PROGRAM PRG_Static
VAR
	k: INT;
	l: INT;
	m: INT;
END_VAR

	stat_scalar_BOOL	:= TRUE;
	stat_scalar_I1		:= 1;	
	stat_scalar_UI1		:= 1;	
	stat_scalar_I2 		:= 1;		
	stat_scalar_UI2		:= 1;	
	stat_scalar_I4		:= 1;	
	stat_scalar_UI4		:= 1;	
	stat_scalar_I8		:= 1;	
	stat_scalar_UI8		:= 1;	
	stat_scalar_BYTE	:= 1;	
	stat_scalar_WORD	:= 1;	
	stat_scalar_DWORD	:= 1;	
	stat_scalar_LWORD	:= 1;				
	stat_scalar_R4		:= 1.0;				
	stat_scalar_R8		:= 1.0;				
	stat_scalar_BSTR	:= 'Hello World';
	stat_scalar_WSTRING	:= "Hello World";
	stat_scalar_DT		:= DT#1972-03-29-00:00:00;
	stat_scalar_DATE 	:= DATE#1972-03-29;
	stat_scalar_TOD		:= TOD#12:00:00;	
	stat_scalar_TIME	:= T#1S;	

	GVL_structures.StructuredType1.a 			:= 42;
	GVL_structures.StructuredType1.b			:= 42;
	GVL_structures.StructuredType1.x			:= E_Enum_1.THREE;
	GVL_structures.StructuredType1.str			:= 'Hello World';

	GVL_structures.StructuredType2.c1.a			:= 42;
	GVL_structures.StructuredType2.c1.b			:= 42;
	GVL_structures.StructuredType2.c1.x			:= E_Enum_1.THREE;
	GVL_structures.StructuredType2.c1.str		:= 'Hello World';
	GVL_structures.StructuredType2.s_5			:= 'Hello';
	GVL_structures.StructuredType2.s_3			:= 'Hel';
	FOR k:= 0 TO 5 DO
		GVL_structures.StructuredType2.cArr[k].a:= 42;
		GVL_structures.StructuredType2.cArr[k].b:= 42;
		GVL_structures.StructuredType2.cArr[k].x:= E_Enum_1.THREE;
		GVL_structures.StructuredType2.cArr[k].str:= 'Hello World'; 
	END_FOR	
	GVL_structures.StructuredType2.e			:= E_Enum_1.THREE;
	FOR k:= 0 TO 100 DO
		GVL_structures.StructuredType2.iArr[k] := 42;
	END_FOR
	
	GVL_structures.StructuredType8.stComplex.a			:= 42;
	GVL_structures.StructuredType8.stComplex.b			:= 42;
	GVL_structures.StructuredType8.stComplex.x			:= E_Enum_1.THREE;
	GVL_structures.StructuredType8.stComplex.str		:= 'Hello World';
	GVL_structures.StructuredType8.strString5			:= 'Hello';
	GVL_structures.StructuredType8.strString3			:= 'Hel';
	FOR k:= 0 TO 1 DO
		GVL_structures.StructuredType8.arrComplex[k].a:= 42;
		GVL_structures.StructuredType8.arrComplex[k].b:= 42;
		GVL_structures.StructuredType8.arrComplex[k].x:= E_Enum_1.THREE;
		GVL_structures.StructuredType8.arrComplex[k].str:= 'Hello World'; 
	END_FOR	
	GVL_structures.StructuredType8.eEnum			:= E_Enum_1.THREE;
	FOR k:= 0 TO 100 DO
		GVL_structures.StructuredType8.arrDint[k] := 42;
	END_FOR	
	
	FOR k:= 0 TO ARRSIZEX DO
		stat_1dim_BOOL[k] := TRUE;
		stat_1dim_I1[k] := 1;
		stat_1dim_UI1[k] := 1;
		stat_1dim_I2[k] := 1;
		stat_1dim_UI2[k] := 1;
		stat_1dim_I4[k] := 1;
		stat_1dim_UI4[k] := 1;
		stat_1dim_I8[k] := 1;
		stat_1dim_UI8[k] := 1;
		stat_1dim_BYTE[k] := 1;
		stat_1dim_WORD[k] := 1;
		stat_1dim_DWORD[k] := 1;
		stat_1dim_LWORD[k] := 1;
		stat_1dim_R4[k] := 1.0;
		stat_1dim_R8[k] := 1.0;
		stat_1dim_BSTR[k] := 'Hello World';
		stat_1dim_WSTRING[k] := "Hello World";
		stat_1dim_DT[k] := DT#1972-03-29-00:00:00;
		stat_1dim_DATE[k] := DATE#1972-03-29;
		stat_1dim_TOD[k] := TOD#12:00:00;
		stat_1dim_TIME[k] := T#1S;
	END_FOR	

FOR l:= 0 TO ARRSIZEY DO
	FOR k:= 0 TO ARRSIZEX DO
		stat_2dim_BOOL[k,l] := TRUE;
		stat_2dim_I1[k,l] := 1;
		stat_2dim_UI1[k,l] := 1;
		stat_2dim_I2[k,l] := 1;
		stat_2dim_UI2[k,l] := 1;
		stat_2dim_I4[k,l] := 1;
		stat_2dim_UI4[k,l] := 1;
		stat_2dim_I8[k,l] := 1;
		stat_2dim_UI8[k,l] := 1;
		stat_2dim_BYTE[k,l] := 1;
		stat_2dim_WORD[k,l] := 1;
		stat_2dim_DWORD[k,l] := 1;
		stat_2dim_LWORD[k,l] := 1;
		stat_2dim_R4[k,l] := 1.0;
		stat_2dim_R8[k,l] := 1.0;
		stat_2dim_BSTR[k,l] := 'Hello World';
		stat_2dim_WSTRING[k,l] := "Hello World";
		stat_2dim_DT[k,l] := DT#1972-03-29-00:00:00;
		stat_2dim_DATE[k,l] := DATE#1972-03-29;
		stat_2dim_TOD[k,l] := TOD#12:00:00;
		stat_2dim_TIME[k,l] := T#1S;
	END_FOR
END_FOR	

FOR m:= 0 TO ARRSIZEY DO
	FOR l:= 0 TO ARRSIZEY DO
		FOR k:= 0 TO ARRSIZEX DO
			stat_3dim_BOOL[k,l,m] := TRUE;
			stat_3dim_I1[k,l,m] := 1;
			stat_3dim_UI1[k,l,m] := 1;
			stat_3dim_I2[k,l,m] := 1;
			stat_3dim_UI2[k,l,m] := 1;
			stat_3dim_I4[k,l,m] := 1;
			stat_3dim_UI4[k,l,m] := 1;
			stat_3dim_I8[k,l,m] := 1;
			stat_3dim_UI8[k,l,m] := 1;
			stat_3dim_BYTE[k,l,m] := 1;
			stat_3dim_WORD[k,l,m] := 1;
			stat_3dim_DWORD[k,l,m] := 1;
			stat_3dim_LWORD[k,l,m] := 1;
			stat_3dim_R4[k,l,m] := 1.0;
			stat_3dim_R8[k,l,m] := 1.0;
			stat_3dim_BSTR[k,l,m] := 'Hello World';
			stat_3dim_WSTRING[k,l,m] := "Hello World";
			stat_3dim_DT[k,l,m] := DT#1972-03-29-00:00:00;
			stat_3dim_DATE[k,l,m] := DATE#1972-03-29;
			stat_3dim_TOD[k,l,m] := TOD#12:00:00;
			stat_3dim_TIME[k,l,m] := T#1S;			
		END_FOR
	END_FOR
END_FOR

END_PROGRAM

(* stored: Version 1.1.0.1, ProductVersion 3.1.4024.0
   POU PRG_Static: Id {b0e82972-5ed0-43dd-ad1d-5023445ae7be}, SpecialFunc None *)
